// This function has been automatically generated from the project information.
{attribute 'signature_flag' := '1073741824'}
{attribute 'TcGenerated'}
{attribute 'no-analysis'}
FUNCTION F_GetCompany : WSTRING
VAR_INPUT
	
END_VAR

F_GetCompany := "Beckhoff Automation LLC";

END_FUNCTION

(* stored: Version 1.1.0.1
   POU F_GetCompany: Id {1c12ce69-4e2d-0d53-1cd8-92e7a1b0e8ea}, SpecialFunc None *)
